// Mitsubishi GX Works2 project: 30   PLC: FX3G

// task Task_01 (event TRUE, interval 0, priority 31): POU_01

PROGRAM POU_01
VAR
  wstep : INT;
END_VAR
M99 := FALSE AND
M4 AND M5 AND M6 AND M7 AND
Y1 AND Y2 AND Y3;

IF M8002 THEN
    wstep := 0;
END_IF;

Y3 := M7;

CASE wstep OF
    0:
        Y1 := M5;
        Y2 := M6 AND (NOT M7);

        IF M4 THEN
            wstep := 1;
        END_IF;
    1:
        Y1 := FALSE;
        Y2 := FALSE;

        IF NOT M4 THEN
            wstep := 0;
        END_IF;
        IF M5 THEN
            wstep := 20;
        END_IF;
        IF M6 AND (NOT M7) THEN
            wstep := 40;
        END_IF;

    20:
        Y1 := TRUE;

        IF NOT M4 THEN
            wstep := 0;
        END_IF;

    40:
        Y2 := TRUE;
        
        IF (NOT M4) OR M7 THEN
            wstep := 0;
        END_IF;
END_CASE;
END_PROGRAM
